// Mitsubishi GX Works2 project: servo2   PLC: Q03UDV

PROGRAM MAIN
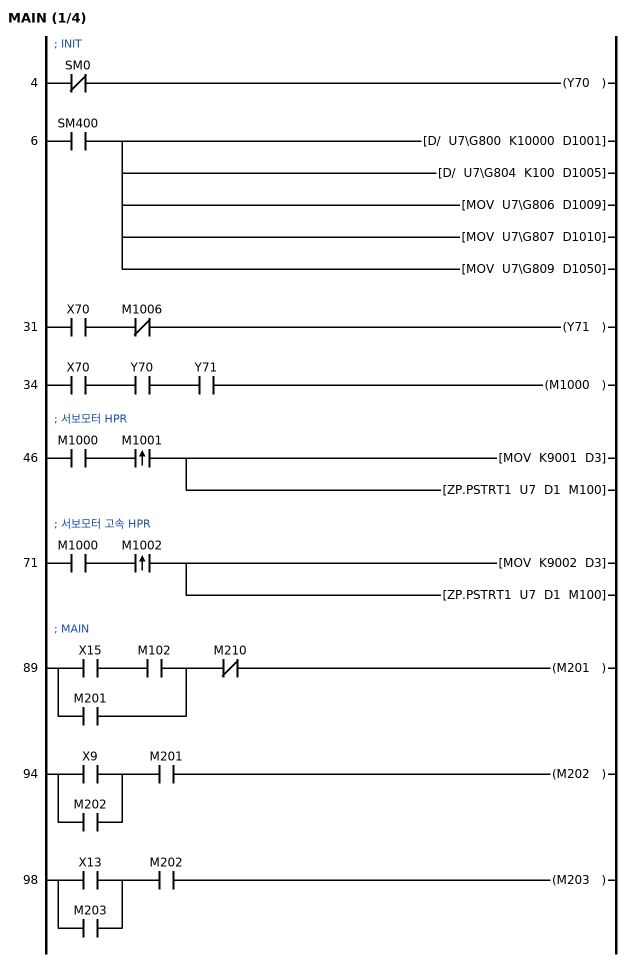
; INIT
4     LDI     SM0
      OUT     Y70
6     LD      SM400
      D/      U7\G800 K10000 D1001
      D/      U7\G804 K100 D1005
      MOV     U7\G806 D1009
      MOV     U7\G807 D1010
      MOV     U7\G809 D1050
31    LD      X70
      ANI     M1006
      OUT     Y71
34    LD      X70
      AND     Y70
      AND     Y71
      OUT     M1000
; 서보모터 HPR
46    LD      M1000
      ANDP    M1001
      MOV     K9001 D3
      ZP.PSTRT1 U7 D1 M100
; 서보모터 고속 HPR
71    LD      M1000
      ANDP    M1002
      MOV     K9002 D3
      ZP.PSTRT1 U7 D1 M100
; MAIN
89    LD      X15
      AND     M102
      OR      M201
      ANI     M210
      OUT     M201
94    LD      X9
      OR      M202
      AND     M201
      OUT     M202
98    LD      X13
      OR      M203
      AND     M202
      OUT     M203
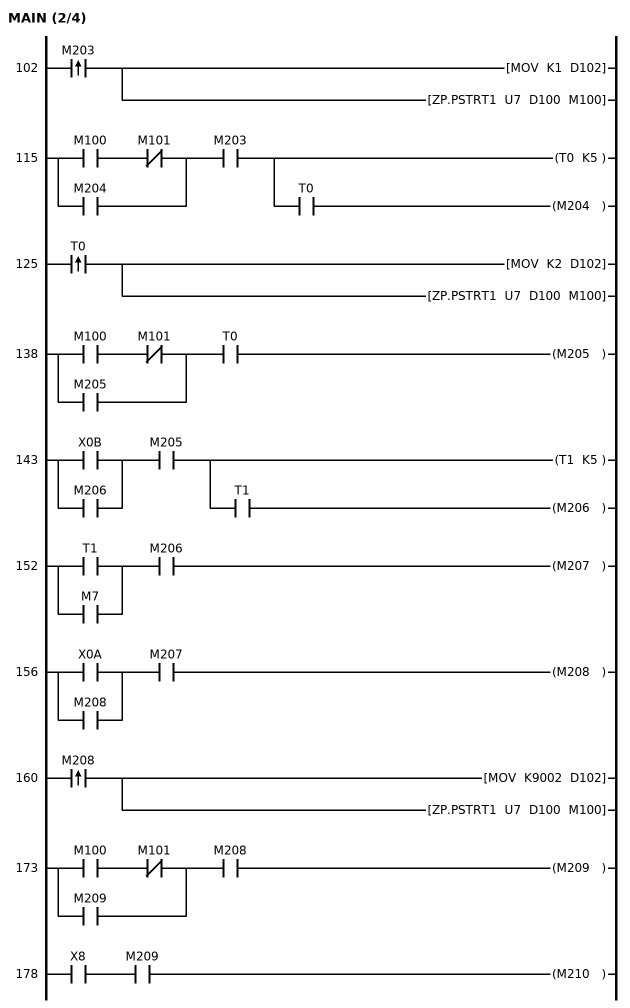
102   LDP     M203
      MOV     K1 D102
      ZP.PSTRT1 U7 D100 M100
115   LD      M100
      ANI     M101
      OR      M204
      AND     M203
      OUT     T0 K5
      AND     T0
      OUT     M204
125   LDP     T0
      MOV     K2 D102
      ZP.PSTRT1 U7 D100 M100
138   LD      M100
      ANI     M101
      OR      M205
      AND     T0
      OUT     M205
143   LD      X0B
      OR      M206
      AND     M205
      OUT     T1 K5
      AND     T1
      OUT     M206
152   LD      T1
      OR      M7
      AND     M206
      OUT     M207
156   LD      X0A
      OR      M208
      AND     M207
      OUT     M208
160   LDP     M208
      MOV     K9002 D102
      ZP.PSTRT1 U7 D100 M100
173   LD      M100
      ANI     M101
      OR      M209
      AND     M208
      OUT     M209
178   LD      X8
      AND     M209
      OUT     M210
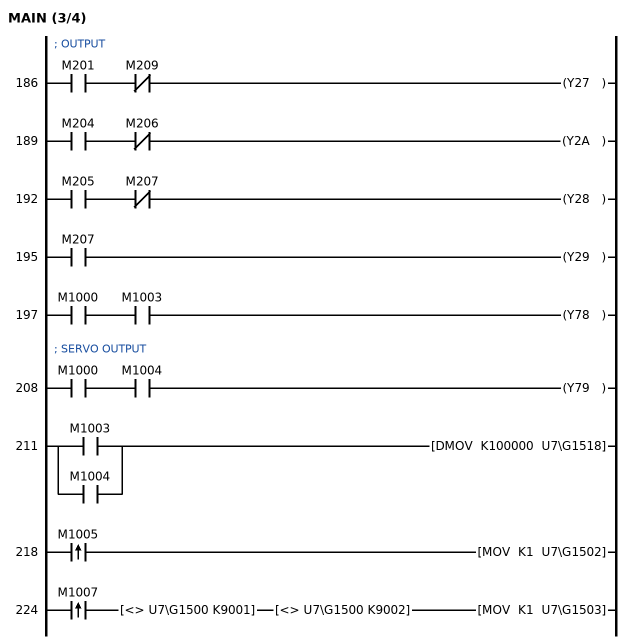
; OUTPUT
186   LD      M201
      ANI     M209
      OUT     Y27
189   LD      M204
      ANI     M206
      OUT     Y2A
192   LD      M205
      ANI     M207
      OUT     Y28
195   LD      M207
      OUT     Y29
197   LD      M1000
      AND     M1003
      OUT     Y78
; SERVO OUTPUT
208   LD      M1000
      AND     M1004
      OUT     Y79
211   LD      M1003
      OR      M1004
      DMOV    K100000 U7\G1518
218   LDP     M1005
      MOV     K1 U7\G1502
224   LDP     M1007
      AND<>   U7\G1500 K9001
      AND<>   U7\G1500 K9002
      MOV     K1 U7\G1503
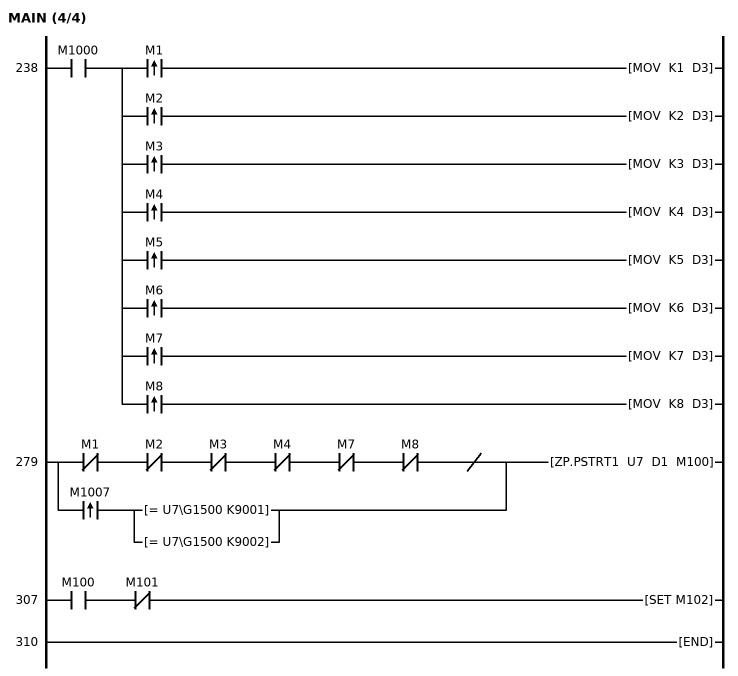
238   LD      M1000
      MPS
      ANDP    M1
      MOV     K1 D3
      MRD
      ANDP    M2
      MOV     K2 D3
      MRD
      ANDP    M3
      MOV     K3 D3
      MRD
      ANDP    M4
      MOV     K4 D3
      MRD
      ANDP    M5
      MOV     K5 D3
      MRD
      ANDP    M6
      MOV     K6 D3
      MRD
      ANDP    M7
      MOV     K7 D3
      MPP
      ANDP    M8
      MOV     K8 D3
279   LDI     M1
      ANI     M2
      ANI     M3
      ANI     M4
      ANI     M7
      ANI     M8
      INV
      LDP     M1007
      LD=     U7\G1500 K9001
      OR=     U7\G1500 K9002
      ANB
      ORB
      ZP.PSTRT1 U7 D1 M100
307   LD      M100
      ANI     M101
      SET     M102
310   END
END_PROGRAM
